// TIA Portal V20 export
DATA_BLOCK "InstE2MenergyMeterDriver"   // DB56
TITLE = Instance of FB E2MenergyMeterDrv
AUTHOR : SICAR
FAMILY : E2M
NAME : E2M_AIEM
VERSION : 2.0
// Energy Meter
// stored: InstanceOfName E2MenergyMeterDrv, InstanceOfType FB
"E2MenergyMeterDrv"
   // VAR_INPUT
   //    id : HW_IO;
   //    firstByteData : Int;
   //    connectionType : Int;
   //    commResourceLimit : Int;
   //    automaticUpdate : Bool;
   //    resetMinMax : Bool;
   //    resetEnergyCounter : Bool;
   //    bitsConnectedHmi : Bool;
   //    backupCycleEnCount : Time;
   // END_VAR
   // VAR_OUTPUT
   //    timeBetweenUpdate : Time;
   //    timeBetweenUpdateMax : Time;
   //    timeStampMeasValues : DTL;
   //    driverData { ExternalAccessible := 'False'; ExternalVisible := 'False'; ExternalWritable := 'False'} : "LSicar_typeEnMeterVisuStruct";
   //    energyCounter { ExternalAccessible := 'False'; ExternalVisible := 'False'; ExternalWritable := 'False'} : "typeEnCounter";
   //    errorCode : DWord;
   //    errorLocation : Word;
   //    timeStampEnCount : DTL;
   // END_VAR
   // VAR_IN_OUT
   //    bitsHmi : "typeEnMeterBits";
   //    commResourceCounter : Int;
   // END_VAR
   // VAR
   //    instReadDataRecord { S7_SetPoint := 'True'} : RDREC;
   //    instWriteDataRecord { S7_SetPoint := 'True'} : WRREC;
   //    instEnCountUpdateTimer { S7_SetPoint := 'True'} : TON_TIME;
   //    instTimeMeasurement { S7_SetPoint := 'True'} : TON_TIME;
   //    instWatchdog { S7_SetPoint := 'True'} : TON_TIME;
   //    statInputVariablesOk : Bool;
   //    statResetEnCountRequest : Bool;
   //    statReadDataRecRequest : Bool;
   //    statWriteDataRecRequest : Bool;
   //    statRestoreEnergy : Bool;
   //    statStartAcyclicHmiOld : Bool;
   //    statResetEnergyHmiOld : Bool;
   //    statResetEnergyOld : Bool;
   //    statResetMinMaxHmiOld : Bool;
   //    statResetMinMaxOld : Bool;
   //    statRunUpdateTimer : Bool;
   //    statWatchdogRun : Bool;
   //    statUserDataVariant : Byte;
   //    statSmState : Int;
   //    statSmStateNext : Int;
   //    statReadRecIndex : Int;
   //    statReadRecMaxLength : UInt;
   //    statTimetoUpdate : Time;
   //    statVmeasurementValues : "typeEnMeterValues";
   //    statVenergyCounter : "typeEnMeterCounter";
   //    statBitsInternalHmi : "typeEnMeterBits";
   // END_VAR
   // VAR RETAIN
   //    statRestoreEnCountValues : "typeEnMeterRestore";
   // END_VAR
   // VAR
   //    statAuxTimeBetweenUpdateMax { S7_SetPoint := 'True'} : Time;
   //    statErrorCode { ExternalVisible := 'False'} : DWord;
   // END_VAR
BEGIN
END_DATA_BLOCK
